KUKA KRL program: placewasher1.src, placewasher1.dat

--- placewasher1.src ---
&ACCESS RVO1
&COMMENT
&ACCESS RVP
&PARAM EDITMASK = *
&PARAM TEMPLATE = C:\KRC\Roboter\Template\vorgabe
&PARAM DISKPATH = KRC:\R1\Program
DEF placewasher1(current_box_layer1:in, Z_pallet:in)
decl int current_box_layer1 ;number of the current layer of boxes at place 1
DECL INT Z_pallet
DECL pos puklwasher, retreat_1_point

; check if there is a requirement to enter the zone from the operator
IF (Entry_Request) THEN
Go_home()
BRAKE
;FOLD WAIT Time= 0.5 sec;%{PE}%R 8.3.22,%MKUKATPBASIS,%CWAIT,%VWAIT,%P 2:0.5
WAIT SEC 0.5
;ENDFOLD
HALT
ENDIF

; movement down in the direction to the pallet place point
;FOLD LIN P1  Vel=2 m/s CPDAT0 Tool[4]:tool_pallet Base[2]:plpallet1;%{PE}%R 8.3.22,%MKUKATPBASIS,%CMOVE,%VLIN,%P 1:LIN, 2:P1, 3:, 5:2, 7:CPDAT0
$BWDSTART=FALSE
LDAT_ACT=LCPDAT0
FDAT_ACT=FP1
BAS(#CP_PARAMS,2)
LIN XP1
;ENDFOLD

; movement to the point above the pallet place point
;FOLD LIN P2 CONT Vel=2.00000 m/s CPDAT2 Tool[4]:tool_pallet Base[2]:plpallet1;%{PE}%R 8.3.22,%MKUKATPBASIS,%CMOVE,%VLIN,%P 1:LIN, 2:P2, 3:C_DIS C_DIS, 5:2.00000, 7:CPDAT2
$BWDSTART=FALSE
LDAT_ACT=LCPDAT2
FDAT_ACT=FP2
BAS(#CP_PARAMS,2.00000)
LIN XP2 C_DIS C_DIS
;ENDFOLD

; coordinates calculation and movement down to place point
xpuklwasher = XP3
xpuklwasher.z = xpuklwasher.z + Z_pallet * (current_box_layer1 - 1)

;FOLD LIN puklpallet Vel=2 m/s CPDAT1 Tool[4]:tool_pallet Base[2]:plpallet1;%{PE}%R 8.3.32,%MKUKATPBASIS,%CMOVE,%VLIN,%P 1:LIN, 2:puklpallet, 3:, 5:2, 7:CPDAT1
$BWDSTART=FALSE
LDAT_ACT=LCPDAT1
FDAT_ACT=Fpuklpallet
BAS(#CP_PARAMS,2)
LIN Xpuklpallet
;ENDFOLD

;FOLD OUT 7 'Vacuum_on'  State= FALSE;%{PE}%R 8.3.22,%MKUKATPBASIS,%COUT,%VOUTX,%P 2:7, 3:Vacuum_on, 5:FALSE, 6:

$OUT[7]=FALSE
;ENDFOLD
;FOLD OUT 8 'Blow'  State= TRUE;%{PE}%R 8.3.22,%MKUKATPBASIS,%COUT,%VOUTX,%P 2:8, 3:Blow, 5:TRUE, 6:

$OUT[8]=TRUE
;ENDFOLD
;FOLD WAIT Time= 0.5 sec;%{PE}%R 8.3.22,%MKUKATPBASIS,%CWAIT,%VWAIT,%P 2:0.5
WAIT SEC 0.5
;ENDFOLD
;FOLD OUT 8 'Blow'  State= FALSE;%{PE}%R 8.3.22,%MKUKATPBASIS,%COUT,%VOUTX,%P 2:8, 3:Blow, 5:FALSE, 6:

$OUT[8]=FALSE
;ENDFOLD
;FOLD WAIT Time= 0.5 sec;%{PE}%R 8.3.22,%MKUKATPBASIS,%CWAIT,%VWAIT,%P 2:0.5
WAIT SEC 0.5
;ENDFOLD
;FOLD OUT 6 'Vacuum_cups'  State= FALSE;%{PE}%R 8.3.22,%MKUKATPBASIS,%COUT,%VOUTX,%P 2:6, 3:Vacuum_cups, 5:FALSE, 6:

$OUT[6]=FALSE
;ENDFOLD

xpuklwasher.z = xpuklwasher.z + 400

; movement up
;FOLD LIN puklwasher CONT Vel=2.00000 m/s CPDAT4 Tool[2]:tool_empty Base[2]:plpallet1;%{PE}%R 8.3.22,%MKUKATPBASIS,%CMOVE,%VLIN,%P 1:LIN, 2:puklwasher, 3:C_DIS C_DIS, 5:2.00000, 7:CPDAT4
$BWDSTART=FALSE
LDAT_ACT=LCPDAT4
FDAT_ACT=Fpuklwasher
BAS(#CP_PARAMS,2.00000)
LIN Xpuklwasher C_DIS C_DIS
;ENDFOLD

;FOLD PTP home  Vel=100 % PDAT5 Tool[2]:tool_empty Base[0];%{PE}%R 8.3.22,%MKUKATPBASIS,%CMOVE,%VPTP,%P 1:PTP, 2:home, 3:, 5:100, 7:PDAT5
$BWDSTART=FALSE
PDAT_ACT=PPDAT5
FDAT_ACT=Fhome
BAS(#PTP_PARAMS,100)
PTP Xhome
;ENDFOLD

END

--- placewasher1.dat ---
&ACCESS RVO1
&COMMENT
DEFDAT placewasher1 PUBLIC
;FOLD EXTERNAL DECLARATIONS;%{PE}%MKUKATPBASIS,%CEXT,%VCOMMON,%P
;FOLD BASISTECH EXT;%{PE}%MKUKATPBASIS,%CEXT,%VEXT,%P
EXT  BAS (BAS_COMMAND  :IN,REAL  :IN )
DECL INT SUCCESS
;ENDFOLD (BASISTECH EXT)
;FOLD USER EXT;%{E}%MKUKATPUSER,%CEXT,%VEXT,%P
;Make here your modifications

;ENDFOLD (USER EXT)
;ENDFOLD (EXTERNAL DECLERATIONS)
; DECL BASIS_SUGG_T LAST_BASIS={POINT1[] "home                    ",POINT2[] "home                    ",CP_PARAMS[] "CPDAT3                  ",PTP_PARAMS[] "PDAT4                   ",CONT[] "                        ",CP_VEL[] "2                       ",PTP_VEL[] "100                     ",SYNC_PARAMS[] "SYNCDAT                 ",SPL_NAME[] "S0                      ",A_PARAMS[] "ADAT0                   "}
DECL E6POS XP1={X 13.9638586,Y -2.41177225,Z 747.639282,A 1.16506231,B 0.0120191490,C 179.989105,S 2,T 3,E1 0.0,E2 0.0,E3 0.0,E4 0.0,E5 0.0,E6 0.0}
DECL FDAT FP1={TOOL_NO 0,BASE_NO 0,IPO_FRAME #BASE,POINT2[] "P1",TQ_STATE FALSE}
DECL LDAT LCPDAT1={VEL 2,ACC 100,APO_DIST 100,APO_FAC 50,AXIS_VEL 100.0,AXIS_ACC 100.0,ORI_TYP #VAR,CIRC_TYP #BASE,JERK_FAC 50.0,GEAR_JERK 50.0,EXAX_IGN 0}
DECL E6POS XP2={X 14.0937529,Y -2.28732562,Z 290.134674,A 1.16510081,B 0.00569414394,C 179.994843,S 2,T 3,E1 0.0,E2 0.0,E3 0.0,E4 0.0,E5 0.0,E6 0.0}
DECL FDAT FP2={TOOL_NO 4,BASE_NO 2,IPO_FRAME #BASE,POINT2[] " ",TQ_STATE FALSE}
DECL LDAT LCPDAT2={VEL 2.00000,ACC 100,APO_DIST 100,APO_FAC 50,AXIS_VEL 100.0,AXIS_ACC 100.0,ORI_TYP #VAR,CIRC_TYP #BASE,JERK_FAC 50.0,GEAR_JERK 50.0,EXAX_IGN 0}
DECL E6POS XP3={X 14.1800137,Y -2.20657802,Z -6.12030271E-05,A 1.16514552,B 1.28041397E-14,C 180.000,S 2,T 3,E1 0.0,E2 0.0,E3 0.0,E4 0.0,E5 0.0,E6 0.0}
DECL LDAT LCPDAT3={VEL 2.00000,ACC 100.000,APO_DIST 100.000,APO_FAC 50.0000,AXIS_VEL 100.000,AXIS_ACC 100.000,ORI_TYP #VAR,CIRC_TYP #BASE,JERK_FAC 50.0000,GEAR_JERK 50.0000,EXAX_IGN 0}
DECL PDAT PPDAT3={VEL 100.000,ACC 100.000,APO_DIST 100.000,GEAR_JERK 50.0000}
DECL E6POS XP4={X 14.1800137,Y -2.20657802,Z 389.601654,A 1.16514552,B 7.20532304E-14,C 180.000,S 2,T 3,E1 0.0,E2 0.0,E3 0.0,E4 0.0,E5 0.0,E6 0.0}
DECL FDAT FP4={TOOL_NO 2,BASE_NO 2,IPO_FRAME #BASE,POINT2[] " ",TQ_STATE FALSE}
DECL LDAT LCPDAT4={VEL 2.00000,ACC 100,APO_DIST 100,APO_FAC 50,AXIS_VEL 100.0,AXIS_ACC 100.0,ORI_TYP #VAR,CIRC_TYP #BASE,JERK_FAC 50.0,GEAR_JERK 50.0,EXAX_IGN 0}
DECL E6POS XP5={X 13.9638586,Y -2.41177225,Z 747.639282,A 1.16506231,B 0.0120191490,C 179.989105,S 2,T 3,E1 0.0,E2 0.0,E3 0.0,E4 0.0,E5 0.0,E6 0.0}
DECL FDAT FP5={TOOL_NO 2,BASE_NO 2,IPO_FRAME #BASE,POINT2[] " ",TQ_STATE FALSE}
DECL PDAT PPDAT5={VEL 100,ACC 100,APO_DIST 100,APO_MODE #CPTP,GEAR_JERK 50}
DECL BASIS_SUGG_T LAST_BASIS={POINT1[] "Home",POINT2[] "P1",CP_PARAMS[] "CPDAT1",PTP_PARAMS[] "PDAT0",CONT[] "",CP_VEL[] "2",PTP_VEL[] "100"}
DECL E6POS Xpuklwasher={X 14.1800137,Y -2.20657802,Z 389.601654,A 1.16514552,B 7.20532304E-14,C 180.000,S 2,T 3,E1 0.0,E2 0.0,E3 0.0,E4 0.0,E5 0.0,E6 0.0}
DECL FDAT Fpuklwasher={TOOL_NO 2,BASE_NO 2,IPO_FRAME #BASE,POINT2[] " ",TQ_STATE FALSE}
ENDDAT
